// SIMATIC S7-200 project (STEP 7-Micro/WIN), CPU 224 AM REL 21.02

ORGANIZATION_BLOCK 主程序:OB1
TITLE=程序注释
BEGIN
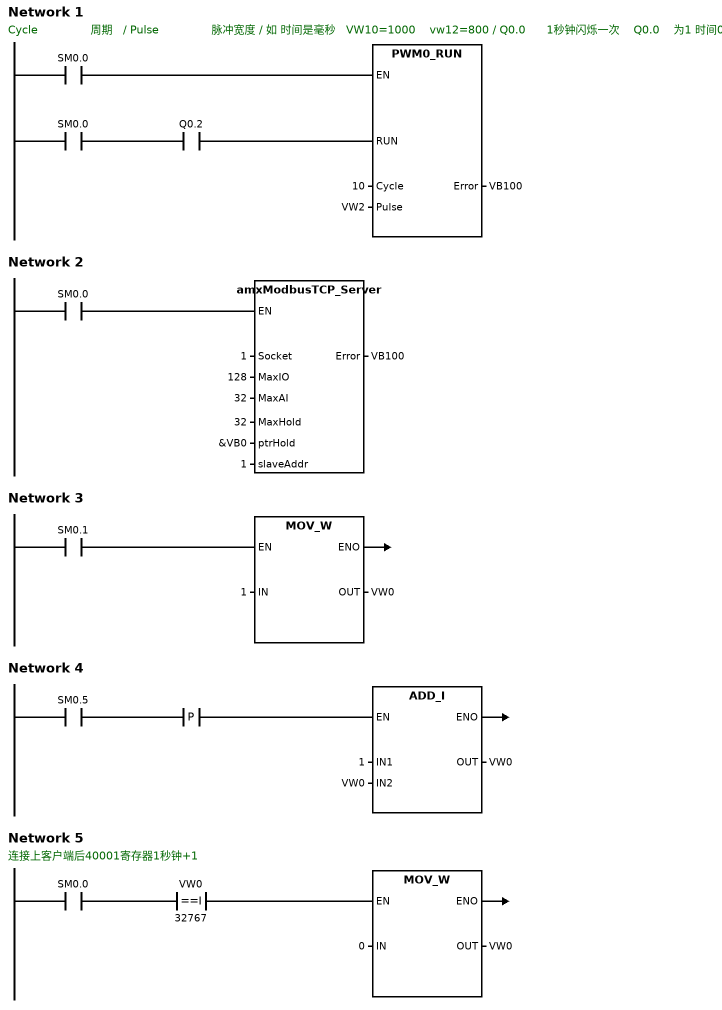
Network 1
// Cycle               周期  
// Pulse               脉冲宽度
// 如 时间是毫秒   VW10=1000    vw12=800
// Q0.0      1秒钟闪烁一次    Q0.0    为1 时间0.8S
LD     SM0.0
=      L60.0
LD     SM0.0
A      Q0.2
=      L63.7
LD     L60.0
CALL   PWM0_RUN:SBR1, L63.7, 10, VW2, VB100
Network 2
LD     SM0.0
CALL   amxModbusTCP_Server:SBR2, 1, 128, 32, 32, &VB0, 1, VB100
Network 3
LD     SM0.1
MOVW   1, VW0
Network 4
LD     SM0.5
EU
+I     1, VW0
Network 5
// 连接上客户端后40001寄存器1秒钟+1
LD     SM0.0
AW=    VW0, 32767
MOVW   0, VW0
END_ORGANIZATION_BLOCK

// SBR1: protected block, not included

SUBROUTINE_BLOCK amxModbusTCP_Server:SBR2
TITLE=子程序注释
VAR_INPUT
Socket:BYTE;	// LB0 1或者2
MaxIO:INT;	// LW1 I 和Q 位最大数目（默认值128）
MaxAI:BYTE;	// LB3 输入寄存器最大数目（模拟输入字-- 16 
MaxHold:BYTE;	// LB4 保持寄存器最大数目（ V 内存字）
ptrHold:DWORD;	// LD5 保持寄存器在V内存中的起始地址（默认值&VB0）
slaveAddr:BYTE;	// LB9 本服务端站号
END_VAR
VAR_OUTPUT
Error:BYTE;	// LB10 错误代码 =1 表示非法的数据地址 ， =2 表示错误的通信口
END_VAR
VAR
tptr:DWORD;	// LD11 
tempa:DWORD;	// LD15 
tempb:INT;	// LW19 
tempc:INT;	// LW21 
END_VAR
BEGIN
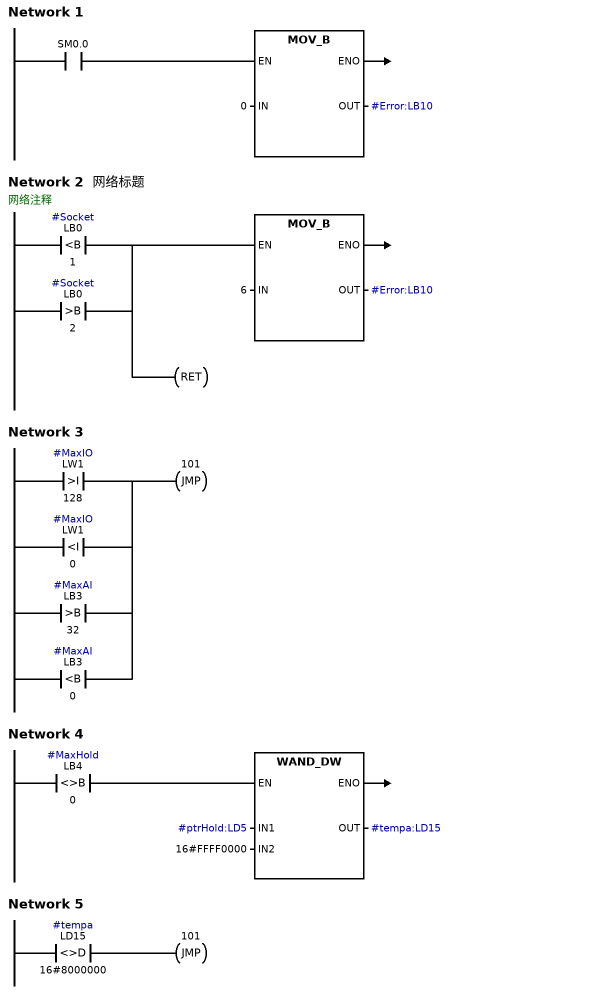
Network 1
LD     SM0.0
MOVB   0, #Error:LB10
Network 2 // 网络标题
// 网络注释
LDB<   #Socket:LB0, 1
OB>    #Socket:LB0, 2
MOVB   6, #Error:LB10
CRET
Network 3
LDW>   #MaxIO:LW1, 128
OW<    #MaxIO:LW1, 0
OB>    #MaxAI:LB3, 32
OB<    #MaxAI:LB3, 0
JMP    101
Network 4
LDB<>  #MaxHold:LB4, 0
MOVD   #ptrHold:LD5, #tempa:LD15
ANDD   16#FFFF0000, #tempa:LD15
Network 5
LDD<>  #tempa:LD15, 16#8000000
JMP    101
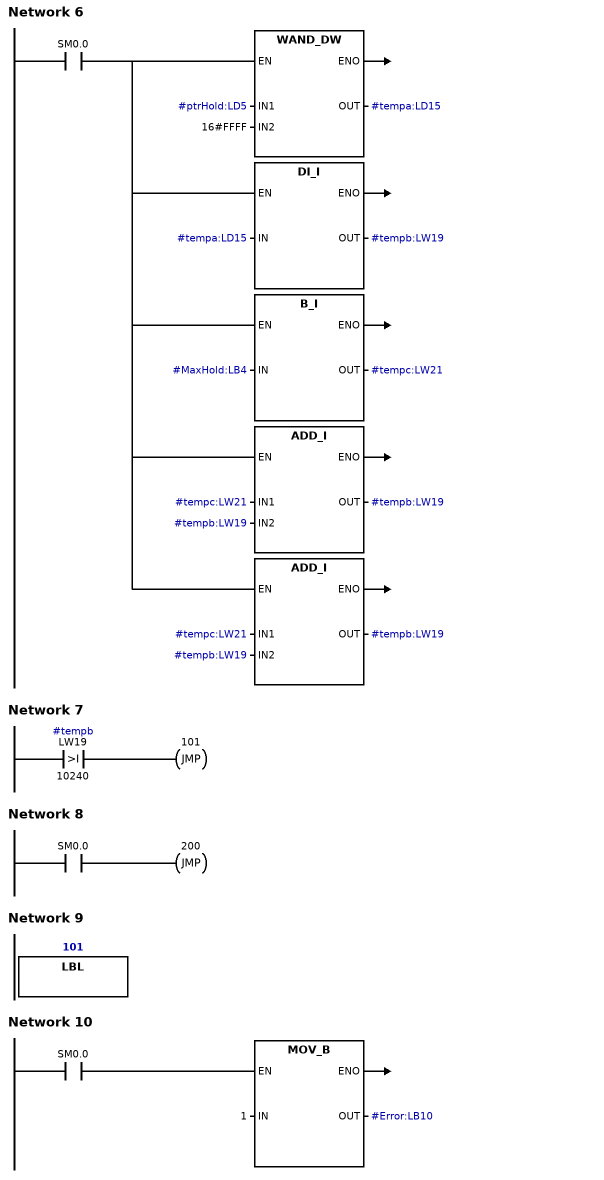
Network 6
LD     SM0.0
MOVD   #ptrHold:LD5, #tempa:LD15
ANDD   16#FFFF, #tempa:LD15
DTI    #tempa:LD15, #tempb:LW19
BTI    #MaxHold:LB4, #tempc:LW21
+I     #tempc:LW21, #tempb:LW19
+I     #tempc:LW21, #tempb:LW19
Network 7
LDW>   #tempb:LW19, 10240
JMP    101
Network 8
LD     SM0.0
JMP    200
Network 9
LBL    101
Network 10
LD     SM0.0
MOVB   1, #Error:LB10
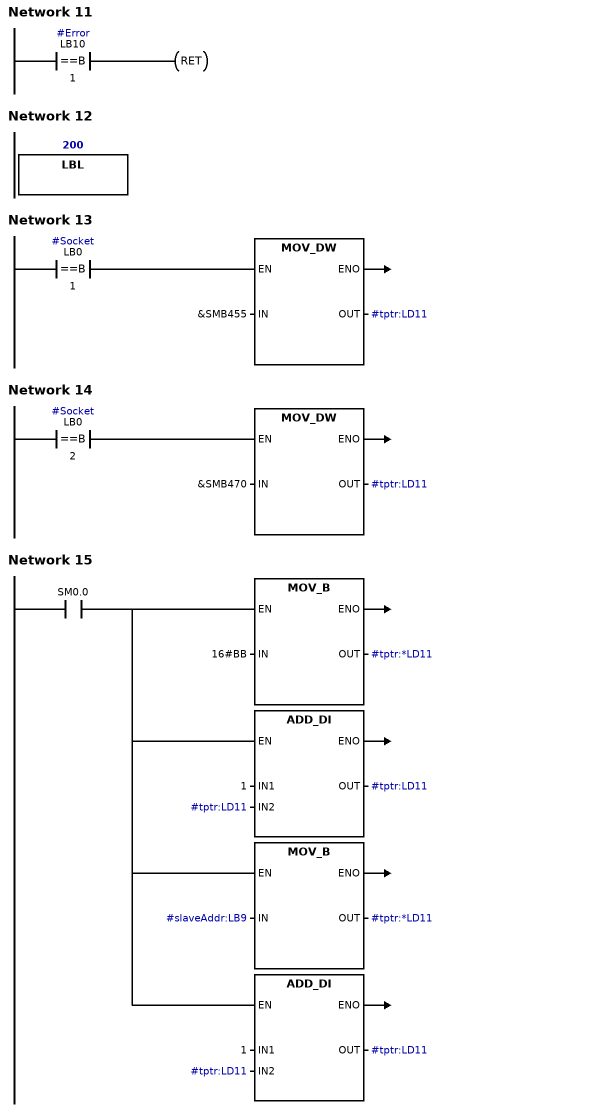
Network 11
LDB=   #Error:LB10, 1
CRET
Network 12
LBL    200
Network 13
LDB=   #Socket:LB0, 1
MOVD   &SMB455, #tptr:LD11
Network 14
LDB=   #Socket:LB0, 2
MOVD   &SMB470, #tptr:LD11
Network 15
LD     SM0.0
MOVB   16#BB, *#tptr:LD11
+D     1, #tptr:LD11
MOVB   #slaveAddr:LB9, *#tptr:LD11
+D     1, #tptr:LD11
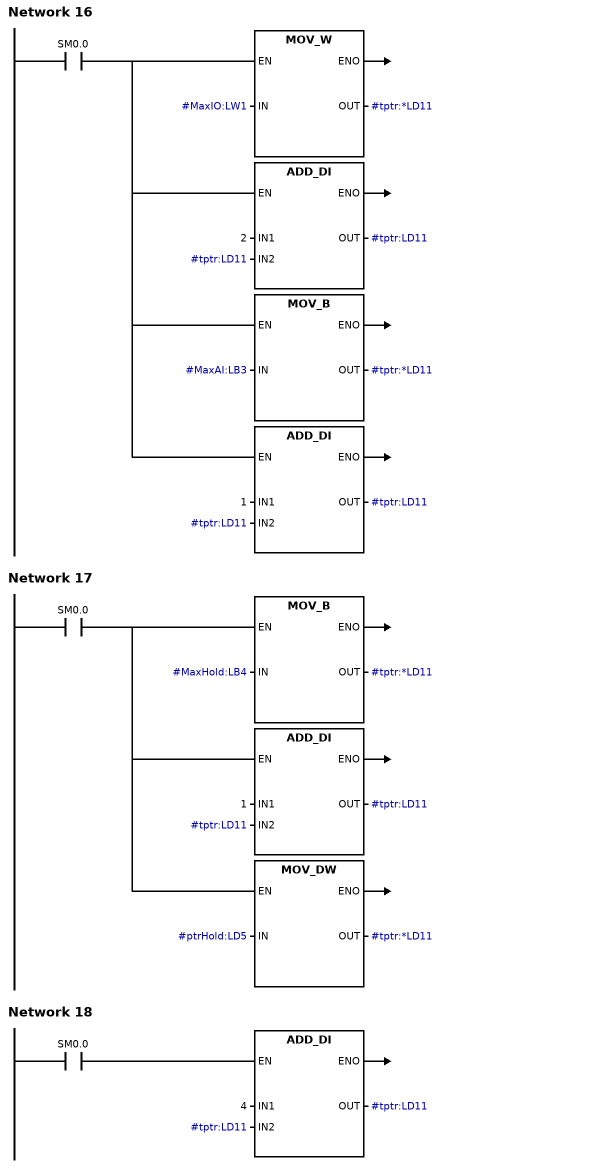
Network 16
LD     SM0.0
MOVW   #MaxIO:LW1, *#tptr:LD11
+D     2, #tptr:LD11
MOVB   #MaxAI:LB3, *#tptr:LD11
+D     1, #tptr:LD11
Network 17
LD     SM0.0
MOVB   #MaxHold:LB4, *#tptr:LD11
+D     1, #tptr:LD11
MOVD   #ptrHold:LD5, *#tptr:LD11
Network 18
LD     SM0.0
+D     4, #tptr:LD11
END_SUBROUTINE_BLOCK

SUBROUTINE_BLOCK MODBUS_TCP_服务器:SBR11
TITLE=
VAR_INPUT
mSlave:BYTE;	// LB0 
mIQ:BYTE;	// LB1 
mInput:BYTE;	// LB2 
mHolding:BYTE;	// LB3 
mAckPtr:DWORD;	// LD4 
END_VAR
BEGIN
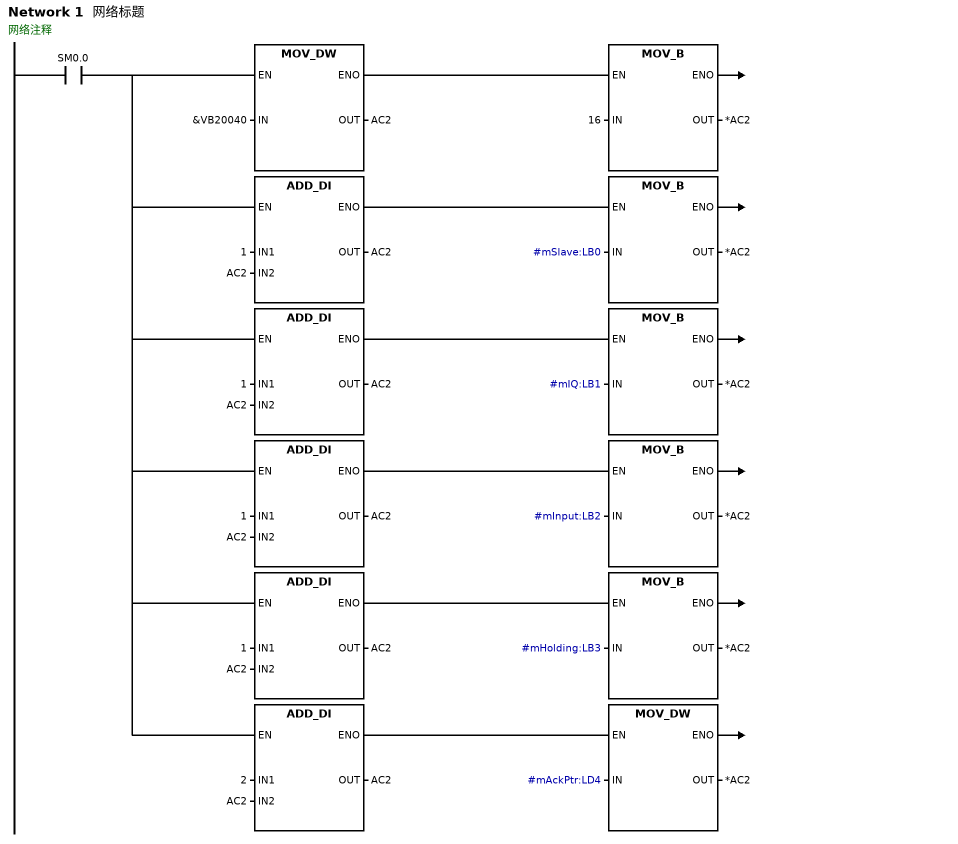
Network 1 // 网络标题
// 网络注释
LD     SM0.0
LPS
MOVD   &VB20040, AC2
AENO
MOVB   16, *AC2
LRD
+D     1, AC2
AENO
MOVB   #mSlave:LB0, *AC2
LRD
+D     1, AC2
AENO
MOVB   #mIQ:LB1, *AC2
LRD
+D     1, AC2
AENO
MOVB   #mInput:LB2, *AC2
LRD
+D     1, AC2
AENO
MOVB   #mHolding:LB3, *AC2
LPP
+D     2, AC2
AENO
MOVD   #mAckPtr:LD4, *AC2
END_SUBROUTINE_BLOCK
